// TIA Portal project "Project1" (V14)

(* hardware
DEVICE "S7-1200 station_1"  S7-1200 Station
   slot 0: "Rack_0"  Rack  V1.0
   slot 1: "PLC_1"  CPU 1214C DC/DC/DC  6ES7 214-1AG40-0XB0  V4.0
*)

// ===== PLC "PLC_1"  CPU 1214C DC/DC/DC =====

VAR_GLOBAL   // PLC tag table "Default tag table"
   "Tag_1" AT %I0.0 : Bool;
   "Tag_2" AT %Q0.0 : Bool;
   "Tag_3" AT %Q0.4 : Bool;
   "Tag_4" AT %Q0.5 : Bool;
   "Tag_5" AT %I0.1 : Bool;
   "Tag_6" AT %Q0.7 : Bool;
   "Tag_7" AT %Q0.2 : Bool;
   "Tag_8" AT %Q0.1 : Bool;
   "Tag_9" AT %Q0.3 : Bool;
   "Tag_10" AT %Q0.6 : Bool;
END_VAR

ORGANIZATION_BLOCK "Main"   // OB1, LAD, ProgramCycle
TITLE = "Main Program Sweep (Cycle)"
{ S7_Optimized_Access := 'TRUE' }
VERSION : 0.1
   VAR_INPUT
      Initial_Call : Bool;   // Initial call of this OB
      Remanence : Bool;   // =True, if remanent data are available
   END_VAR
BEGIN

REGION Network 1
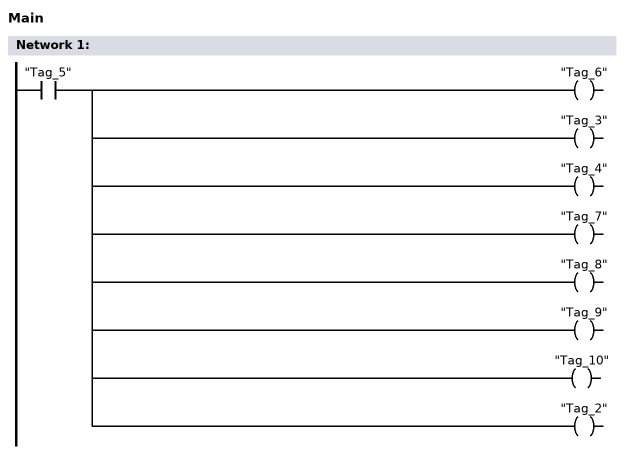
   RUNG wire#powerrail
      Contact( "Tag_5" )
      wire#w1
      Coil( "Tag_6" )
   END_RUNG
   RUNG wire#w1
      Coil( "Tag_3" )
   END_RUNG
   RUNG wire#w1
      Coil( "Tag_4" )
   END_RUNG
   RUNG wire#w1
      Coil( "Tag_7" )
   END_RUNG
   RUNG wire#w1
      Coil( "Tag_8" )
   END_RUNG
   RUNG wire#w1
      Coil( "Tag_9" )
   END_RUNG
   RUNG wire#w1
      Coil( "Tag_10" )
   END_RUNG
   RUNG wire#w1
      Coil( "Tag_2" )
   END_RUNG
   // the same network as SCL:
   "Tag_6" := "Tag_5";
   "Tag_3" := "Tag_5";
   "Tag_4" := "Tag_5";
   "Tag_7" := "Tag_5";
   "Tag_8" := "Tag_5";
   "Tag_9" := "Tag_5";
   "Tag_10" := "Tag_5";
   "Tag_2" := "Tag_5";
END_REGION
END_ORGANIZATION_BLOCK